# EPICS autosave request: iocs/voxtelIOC/iocBoot/iocVoxtel/auto_settings.req
file "voxtel_settings.req",        P=$(P),  R=cam1:
#file "NDFileRaw_settings.req",        P=$(P),  R=raw1:
file "NDStdArrays_settings.req",  P=$(P),  R=image1:
file "commonPlugin_settings.req", P=$(P)
